INTERFACE IPAScale EXTENDS IACComponent

END_INTERFACE

(* stored: Version 1.1.0.1, ProductVersion 3.1.4020.12
   Itf IPAScale: Id {990f2d21-6f1a-4b74-9f5e-d50565462be6} *)
